(* CODESYS project ESME_Git_Test
   Author: SEDK
   Title: Untitled5
   Version: 0.0.0.0

Project tree, tasks and I/O mapping:
  MyController : TM262L10MESE8T, Schneider Electric, order no. TM262L10MESE8T, version 5.2.8.4
    application Application
      task MAST (cyclic, interval 10 ms, priority 15, watchdog 50 ms x 1) calls SR_Main
      function block BWork1 [FBD]
      function block bWork2 [FBD]
      EM01/
        data type EM01_Data
        function block EM_01 [ST]
      global variables GVL
      function block MyFeature670 [FBD]
      function block MyNewFeature400 [FBD]
      function block New_Branch [FBD]
      function block POU_1 [LD]
      program POU [LD]
      program SR_Feature [LD]
      program SR_Main [ST]
    Diagnostic
    Machine Assistant
    Message Logger
    COM_Bus : COM Bus - TMS, Schneider Electric, version 5.2.8.4
    DI : Digital Inputs, Schneider Electric, version 5.2.8.4
        input  ibDI_IB0 : BYTE  // IB0
        input  ibDI_IB1 : BYTE  // IB1
    DQ : Digital Outputs, Schneider Electric, version 5.2.8.4
        output qbDQ_QB0 : BYTE  // QB0
        output qbDQ_QB1 : BYTE  // QB1
    Ethernet_1 : ETH1, Schneider Electric, version 5.2.8.4
    Ethernet_2 : ETH2, Schneider Electric, version 5.2.8.4
    IO_Bus : IO bus - TM3, Schneider Electric, version 5.2.8.4
    Serial_Line : Serial line, Schneider Electric, version 5.2.8.4
      Machine_Expert_Network_Manager : Machine Expert-Network Manager, Schneider Electric, version 4.0.0.4
  function GetTextProperty2 [ST]
  function GetTextProperty [ST]
  function GetTitle [ST]
*)

// MyController/Application/EM01/EM01_Data
TYPE EM01_Data :
STRUCT
	Data1 : BOOL;
END_STRUCT
END_TYPE

// MyController/Application/GVL
{attribute 'qualified_only'}
VAR_GLOBAL
END_VAR

// MyController/Application/SR_Main
PROGRAM SR_Main
VAR
END_VAR

END_PROGRAM

// GetTextProperty2
// This function has been automatically generated from the project information.
{attribute 'signature_flag' := '1073741824'}
{attribute 'register_in_runtime'}
FUNCTION GetTextProperty2 : POINTER TO WSTRING
VAR_INPUT
	stKey: WSTRING;
END_VAR

IF stKey = "Author" THEN
	GetTextProperty2 := ADR("SEDK");
ELSIF stKey = "Company" THEN
	GetTextProperty2 := ADR("");
ELSIF stKey = "Description" THEN
	GetTextProperty2 := ADR("");
ELSIF stKey = "Project" THEN
	GetTextProperty2 := ADR("Untitled5");
ELSIF stKey = "Title" THEN
	GetTextProperty2 := ADR("Untitled5");
ELSE
	GetTextProperty2 := ADR("");
END_IF

END_FUNCTION

// GetTextProperty
// This function has been automatically generated from the project information.
{attribute 'signature_flag' := '1073741824'}
{attribute 'register_in_runtime'}
FUNCTION GetTextProperty : WSTRING
VAR_INPUT
	stKey: WSTRING;
END_VAR

IF stKey = "Author" THEN
	GetTextProperty := "SEDK";
ELSIF stKey = "Company" THEN
	GetTextProperty := "";
ELSIF stKey = "Description" THEN
	GetTextProperty := "";
ELSIF stKey = "Project" THEN
	GetTextProperty := "Untitled5";
ELSIF stKey = "Title" THEN
	GetTextProperty := "Untitled5";
ELSE
	GetTextProperty := "";
END_IF

END_FUNCTION

// GetTitle
// This function has been automatically generated from the project information.
{attribute 'signature_flag' := '1073741824'}
{attribute 'register_in_runtime'}
FUNCTION GetTitle : WSTRING
VAR_INPUT
	
END_VAR

GetTitle := "Untitled5";

END_FUNCTION

// MyController/Application/BWork1
FUNCTION_BLOCK BWork1
VAR_INPUT
END_VAR
VAR_OUTPUT
END_VAR
VAR
END_VAR

// NETWORK 1

END_FUNCTION_BLOCK

// MyController/Application/bWork2
FUNCTION_BLOCK bWork2
VAR_INPUT
END_VAR
VAR_OUTPUT
END_VAR
VAR
END_VAR

// NETWORK 1

END_FUNCTION_BLOCK

// MyController/Application/MyFeature670
FUNCTION_BLOCK MyFeature670
VAR_INPUT
END_VAR
VAR_OUTPUT
END_VAR
VAR
END_VAR

// NETWORK 1

END_FUNCTION_BLOCK

// MyController/Application/MyNewFeature400
FUNCTION_BLOCK MyNewFeature400
VAR_INPUT
END_VAR
VAR_OUTPUT
END_VAR
VAR
END_VAR

// NETWORK 1

END_FUNCTION_BLOCK

// MyController/Application/New_Branch
FUNCTION_BLOCK New_Branch
VAR_INPUT
END_VAR
VAR_OUTPUT
END_VAR
VAR
END_VAR

// NETWORK 1

END_FUNCTION_BLOCK

// MyController/Application/POU_1
FUNCTION_BLOCK POU_1
VAR_INPUT
END_VAR
VAR_OUTPUT
END_VAR
VAR
END_VAR

// NETWORK 1

END_FUNCTION_BLOCK

// MyController/Application/POU
PROGRAM POU
VAR
END_VAR

// NETWORK 1

END_PROGRAM

// MyController/Application/SR_Feature
PROGRAM SR_Feature
VAR
	xCoil: BOOL;
END_VAR

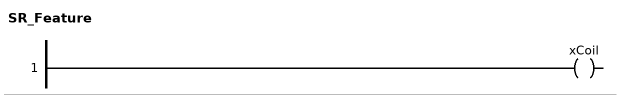
// NETWORK 1
xCoil := TRUE;

END_PROGRAM

// MyController/Application/EM01/EM_01
FUNCTION_BLOCK EM_01
VAR_INPUT
END_VAR
VAR_OUTPUT
END_VAR
VAR
	Myloop: INT;
END_VAR

// Code block1 
Myloop := Myloop+1;


// Code block2
Myloop := Myloop+1;

END_FUNCTION_BLOCK
